Staubli VAL3: USERPAGE.dtx

bool Show
bool bReadWrite[9]
  [0] = true
  [1] = true
  [2] = true
  [3] = true
  [4] = true
  [5] = true
  [6] = true
  [7] = true
  [8] = true
public bool bShowDialog
public bool bUseEscape
public bool bUseRefresh
public num nBottomX[2]
  [0] = 38
  [1] = 38
public num nBottomY = 12
num nFirst
num nKey = 270
num nOffSet
num nOldValue[2]
  [0] = 200
  [1] = 200
public num nPage = 100000
public num nParaAdjustType
num nTest
public num nToSuperV = -1
public num nTopX[2]
public num nTopY
public num nView
public string sItems[9]
  [0] = "使用真空压力传感器    > true "
  [1] = "传送带调速            > false"
  [2] = "距离上限距离1         > -110 mm"
  [3] = "距离上限距离2         > 20 mm"
  [4] = "Bypass个数            > 0"
  [5] = "Bypass前距离上限的距离> -200 mm"
  [6] = "沿传送带X方向偏移     > 0 mm"
  [7] = "沿传送带Y方向偏移     > 0 mm"
  [8] = "沿传送带Z方向偏移     > 0 mm"
string sMessage
public string sTitle = "出料传送带设置"
public string sToSuperV
string stest[11]
  [0] = "sbx"
  [1] = "sdfgsd"
  [2] = "bsfghsfh"
  [3] = "sdfgsdfg"
  [4] = "shsgh"
  [5] = "ghdfh"
  [6] = "snsfg"
  [7] = "sfgsg"
  [8] = "sfgsdfg"
  [9] = "sfgs"
  [10] = "dfsgs"
string stest2
string stest3
